FUNCTION_BLOCK "SCL"
{ S7_Optimized_Access := 'TRUE' }
VERSION : 0.1

BEGIN
END_FUNCTION_BLOCK

